(* CODESYS project CUS-1929

Project tree, tasks and I/O mapping:
  Device : CODESYS Control for PLCnext SL, CODESYS GmbH, order no. 2302000033, version 4.9.0.0
    application Application
      libraries: Standard, 3.5.18.0 (System)
      task MainTask (cyclic, interval t#4ms, priority 1) calls PLC_PRG
      program PLC_PRG [ST]
    PLCNext_Axioline : PLCNext Axioline, CODESYS GmbH, order no. 1068857, version 4.9.0.0
    SoftMotion General Axis Pool
*)

// Device/Application/PLC_PRG
PROGRAM PLC_PRG
VAR
END_VAR

END_PROGRAM
